FUNCTION_BLOCK Test_TStreamAdd_Read_REAL EXTENDS TUnitTestBase
VAR
    Stream : TStream(StreamLength := 2);
END_VAR



Stream.Init(2);

Stream.Add_REAL(1.234567);
    
Assertion.AssertEquals_UDINT(
    Expected := 4,
    Actual := Stream.Position,
    VariableName := 'Stream.Position');
    
Stream.Seek(0);

Assertion.AssertEquals_REAL(
    Expected := 1.234567,
    Actual := Stream.Read_REAL(),
    Delta  := 0.000001,
    VariableName := 'Stream.Read_REAL()');
    
Assertion.AssertEquals_UDINT(
    Expected := 4,
    Actual := Stream.Position,
    VariableName := 'Stream.Position');
    
    
TestFinished();

END_FUNCTION_BLOCK

(* stored: Version 1.1.0.1, ProductVersion 3.1.4024.4
   POU Test_TStreamAdd_Read_REAL: Id {f6f24f4f-449f-4d4b-9188-09f3d21a95c8}, SpecialFunc None *)
